NETWORK
TITLE =EA14_V41
// Act 016
// Box           : VSA14
// Input address : I96.2
// Output address: Q96.2
      CALL FC    70 (
           UnitNo                   := #UnitNo,
           ActRec                   := DB5140.EA14_V41,
           Typ                      := 1,
           FBa                      := #xTmp,
           FBa2                     := I     96.2,
           Out                      := Q     96.2);

NETWORK
TITLE =EA14_V42
// Act 017
// Box           : VSA14
// Input address : I96.3
// Output address: Q96.3
      CALL FC    70 (
           UnitNo                   := #UnitNo,
           ActRec                   := DB5140.EA14_V42,
           Typ                      := 1,
           FBa                      := #xTmp,
           FBa2                     := I     96.3,
           Out                      := Q     96.3);

NETWORK
TITLE =A14_START_MOLCH_LDT
// Act 019
// Box           : VSA14
// Output address: Q98.7
      CALL FC    70 (
           UnitNo                   := #UnitNo,
           ActRec                   := DB5140.A14_START_MOLCH_LDT,
           Typ                      := 0,
           FBa                      := #xTmp,
           FBa2                     := #xTmp,
           Out                      := Q     98.7);

NETWORK
TITLE =Molch ist unterwegs (Mixer)


      CALL FC    70 (
           UnitNo                   := #UnitNo,
           ActRec                   := DB5140.Act20,
           Typ                      := 0,
           FBa                      := #xTmp,
           FBa2                     := #xTmp,
           Out                      := Q    911.5);

NETWORK
TITLE =Molch in Endposition (Mixer)


      CALL FC    70 (
           UnitNo                   := #UnitNo,
           ActRec                   := DB5140.Act21,
           Typ                      := 0,
           FBa                      := #xTmp,
           FBa2                     := #xTmp,
           Out                      := Q    912.6);

NETWORK
TITLE =A14_POS_MOLCH
// Act 030
// Box           : VSA14
// Output address: Q98.4
      CALL FC    70 (
           UnitNo                   := #UnitNo,
           ActRec                   := DB5140.A14_POS_MOLCH,
           Typ                      := 0,
           FBa                      := #xTmp,
           FBa2                     := #xTmp,
           Out                      := Q     98.4);

NETWORK
TITLE =A14_LAUFZEIT_MOLCH
// Act 031
// Box           : VSA14
// Output address: Q98.5
      CALL FC    70 (
           UnitNo                   := #UnitNo,
           ActRec                   := DB5140.A14_LAUFZEIT_MOLCH,
           Typ                      := 0,
           FBa                      := #xTmp,
           FBa2                     := #xTmp,
           Out                      := Q     98.5);

NETWORK
TITLE =A14_TEMP_ERREICHT
// Act 032
// Box           : VSA14
// Output address: Q98.6
      CALL FC    70 (
           UnitNo                   := #UnitNo,
           ActRec                   := DB5140.A14_TEMP_ERREICHT,
           Typ                      := 0,
           FBa                      := #xTmp,
           FBa2                     := #xTmp,
           Out                      := Q     98.6);

NETWORK
TITLE =A14_Schwenkbogen  "1"=CIP  "0"=Produktion
// Act 045
// Box           : Sirup
// Output address: DB_SEND_DOEHLER.Anlage14.Schwenkbogen
      CALL FC    70 (
           UnitNo                   := #UnitNo,
           ActRec                   := DB5140.A14_Schwenkbogen,
           Typ                      := 0,
           FBa                      := #xTmp,
           FBa2                     := #xTmp,
           Out                      := DB404.DBX   67.0);

NETWORK
TITLE =A14_Molch_Sirup  "1"=Molch ist im Sirupraum
// Act 046
// Box           : Sirup
// Output address: DB_SEND_DOEHLER.Anlage14.Molch_Sirup
      CALL FC    70 (
           UnitNo                   := #UnitNo,
           ActRec                   := DB5140.A14_Molch_Sirup,
           Typ                      := 0,
           FBa                      := #xTmp,
           FBa2                     := #xTmp,
           Out                      := DB404.DBX   66.0);

NETWORK
TITLE =A14_Molch_Anlage  "1"=Molch ist an der Anlage
// Act 047
// Box           : Sirup
// Output address: DB_SEND_DOEHLER.Anlage14.Molch_Anlage
      CALL FC    70 (
           UnitNo                   := #UnitNo,
           ActRec                   := DB5140.A14_Molch_Anlage,
           Typ                      := 0,
           FBa                      := #xTmp,
           FBa2                     := #xTmp,
           Out                      := DB404.DBX   66.1);

NETWORK
TITLE =A14_Molch_PRO  "1"=Molch ist bereit für Produktion
// Act 048
// Box           : Sirup
// Output address: DB_SEND_DOEHLER.Anlage14.Molch_PRO
      CALL FC    70 (
           UnitNo                   := #UnitNo,
           ActRec                   := DB5140.A14_Molch_PRO,
           Typ                      := 0,
           FBa                      := #xTmp,
           FBa2                     := #xTmp,
           Out                      := DB404.DBX   66.2);

NETWORK
TITLE =A14_Molch_CIP  "1"=Molch ist bereit für CIP
// Act 049
// Box           : Sirup
// Output address: DB_SEND_DOEHLER.Anlage14.Molch_CIP
      CALL FC    70 (
           UnitNo                   := #UnitNo,
           ActRec                   := DB5140.A14_Molch_CIP,
           Typ                      := 0,
           FBa                      := #xTmp,
           FBa2                     := #xTmp,
           Out                      := DB404.DBX   66.3);

NETWORK
TITLE =A14_Sirupanforderung
// Act 050
// Box           : Sirup
// Output address: DB_SEND_DOEHLER.Anlage14.Sirupanforderung
      CALL FC    70 (
           UnitNo                   := #UnitNo,
           ActRec                   := DB5140.A14_Sirupanforderung,
           Typ                      := 0,
           FBa                      := #xTmp,
           FBa2                     := #xTmp,
           Out                      := DB404.DBX   66.4);

END_FUNCTION_BLOCK

FUNCTION_BLOCK FB 4141
TITLE =U114: Transfer Plant 14
FAMILY : BOTEC_F1
NAME : UniE
VERSION : 1.2


VAR_TEMP
  CIP : BOOL ;	//CIP active
  UNIM : BOOL ;	//Unit Not In Maintenance
  GenRel : BOOL ;	//general OK (emergency and maintenance OK)
  EStopOK : BOOL ;	//emergency OK
  UnitNo : INT ;	//unit number
  xTmp : BOOL ;	//Temporary Bool
  iTmp : INT ;	//Temporary INT
  rTmp : REAL ;	//Temporary REAL
  dTmp : DINT ;	//Temporary DINT (free for general use)
  RetValInt : INT ;	//return value
END_VAR
BEGIN
NETWORK
TITLE =General

      SET   ;
// Simulation ---------------------------------------------------------------
      A     DB4141.DBX 1357.7;
      CC    FB  4149; // "U114Sim"
      A     DB4141.DBX   17.3;
      =     DB4141.DBX 1357.7; //Help bit for simulation

// get unit number ----------------------------------------------------------
      L     DB4140.DBW    0;
      T     #UnitNo;

// communication ------------------------------------------------------------
      UC    FB  4145; // U114Com

NETWORK
TITLE =Sequence organisation

      CLR   ;
      =     M    122.2;

// sequencer ----------------------------------------------------------------
      A     DB4143.DBX   43.1;
      S     DB4143.DBX   97.3;

      CALL FC    40 (
           UnitNo                   := #UnitNo);

END_FUNCTION_BLOCK

FUNCTION_BLOCK FB 4210
TITLE =U121: Planung Transfer VE1
FAMILY : BOTEC_F1
NAME : U121A
VERSION : 2.1


VAR_TEMP
  EStopOK : BOOL ;	//auxiliary flag
  CIP : BOOL ;	//CIP Program Selected
  xTmp : BOOL ;	//Temporary Bool(free for general use)
  DummyBool : BOOL ;	//Temporary Bool(free for general use)
  UnitNo : INT ;	//unit number
  UnitFB : INT ;	//unit expansion FB number
  rTmp : REAL ;	//Temporary REAL (free for general use)
  iTmp : INT ;	//Temporary INT (free for general use)
  DummyInt : INT ;	//Temporary INT (free for general use)
  dTmp : DINT ;	//Temporary DINT (free for general use)
END_VAR
BEGIN
NETWORK
TITLE =general

      CLR   ;
      =     #xTmp;
      =     #EStopOK;

      L     DB4210.DBW    0;
      T     #UnitNo;
      L     DB4210.DBW    2;
      T     #UnitFB;

NETWORK
TITLE =analog inputs

      NOP   0;
// C_AnI01 AnI 001 spare
      CALL FC    24 (
           UnitNo                   := #UnitNo,
           AnIRec                   := DB5213.C_AnI01,
           ValPer                   := #DummyInt);

// C_AnI002 AnI 002 spare
      CALL FC    24 (
           UnitNo                   := #UnitNo,
           AnIRec                   := DB5213.C_AnI002,
           ValPer                   := #DummyInt);

// AnI03 AnI 003 spare
      CALL FC    24 (
           UnitNo                   := #UnitNo,
           AnIRec                   := DB5213.AnI03,
           ValPer                   := #DummyInt);

NETWORK
TITLE =Universal value

      NOP   0;
// unv001 UnV 001 Process Status
      CALL FC    27 (
           UnitNo                   := #UnitNo,
           UnVRec                   := DB5215.unv001,
           ValExt                   := DB5215.DBD  234);

// unv002 UnV 002 Universal Value 02
      CALL FC    27 (
           UnitNo                   := #UnitNo,
           UnVRec                   := DB5215.unv002,
           ValExt                   := DB5215.DBD  362);

// unv003 UnV 003 Druck Sollwert
      CALL FC    27 (
           UnitNo                   := #UnitNo,
           UnVRec                   := DB5215.unv003,
           ValExt                   := DB5215.DBD  490);

// unv004 UnV 004 Universal Value 04
      CALL FC    27 (
           UnitNo                   := #UnitNo,
           UnVRec                   := DB5215.unv004,
           ValExt                   := DB5215.DBD  618);

NETWORK
TITLE =special inputs

      NOP   0;
// SpI01 SpI 001 spare
      CALL FC    14 (
           UnitNo                   := #UnitNo,
           SpIRec                   := DB5211.SpI01,
           SpIBit                   := #DummyBool);

// SpI02 SpI 002 spare
      CALL FC    14 (
           UnitNo                   := #UnitNo,
           SpIRec                   := DB5211.SpI02,
           SpIBit                   := #DummyBool);

// SpI03 SpI 003 spare
      CALL FC    14 (
           UnitNo                   := #UnitNo,
           SpIRec                   := DB5211.SpI03,
           SpIBit                   := #DummyBool);

// SpI04 SpI 004 spare
      CALL FC    14 (
           UnitNo                   := #UnitNo,
           SpIRec                   := DB5211.SpI04,
           SpIBit                   := #DummyBool);

NETWORK
TITLE =messages

      NOP   0;
// msg001 Msg 001 Message 01
      CALL FC    16 (
           UnitNo                   := #UnitNo,
           MsgRec                   := DB5217.msg001,
           MsgBit                   := DB5217.DBX   82.7);

// msg002 Msg 002 Message 02
      CALL FC    16 (
           UnitNo                   := #UnitNo,
           MsgRec                   := DB5217.msg002,
           MsgBit                   := DB5217.DBX  142.7);

// msg003 Msg 003 Message 03
      CALL FC    16 (
           UnitNo                   := #UnitNo,
           MsgRec                   := DB5217.msg003,
           MsgBit                   := DB5217.DBX  202.7);

NETWORK
TITLE =controllers

      NOP   0;
// PID01 PID 001 spare
      CALL FC    55 (
           UnitNo                   := #UnitNo,
           PIDRec                   := DB5216.PID01,
           SpExt                    := DB5216.DBD  234,
           PVal                     := DB5216.DBD  254,
           OPer                     := #DummyInt);

NETWORK
TITLE =unit supply

      UC    FB [#UnitFB];
END_FUNCTION_BLOCK

FUNCTION_BLOCK FB 4211
TITLE =U121: Planung Transfer VE1
FAMILY : BOTEC_F1
NAME : U121E
VERSION : 1.2


VAR_TEMP
  CIP : BOOL ;	//CIP active
  UNIM : BOOL ;	//Unit Not In Maintenance
  GenRel : BOOL ;	//general OK (emergency and maintenance OK)
  EStopOK : BOOL ;	//emergency OK
  UnitNo : INT ;	//unit number
  xTmp : BOOL ;	//Temporary Bool
  iTmp : INT ;	//Temporary INT
  rTmp : REAL ;	//Temporary REAL
  dTmp : DINT ;	//Temporary DINT (free for general use)
  RetValInt : INT ;	//return value
END_VAR
BEGIN
NETWORK
TITLE =General

      SET   ;
// Simulation ---------------------------------------------------------------
      A     DB4211.DBX 1357.7;
      CC    FB  4219; // "U121Sim"
      A     DB4211.DBX   17.3;
      =     DB4211.DBX 1357.7; //Help bit for simulation

// get unit number ----------------------------------------------------------
      L     DB4210.DBW    0;
      T     #UnitNo;

// CIP ----------------------------------------------------------------------
      L     DB4211.DBD   54;
      L     0;
      <D    ;
      =     #CIP;

// emergency OK -------------------------------------------------------------
      A     DB4215.DBX   27.0; //Emergency Stop OK
      =     #EStopOK;

// Write Unit in Maintenance ------------------------------------------------

      AN    DB4211.DBX   69.7;
      =     #UNIM;

// emergency and maintenance OK ---------------------------------------------
      A     #EStopOK;
      A     #UNIM;
      =     #GenRel;

// communication ------------------------------------------------------------
      UC    FB  4215; // U121Com

NETWORK
TITLE =Analog Inputs

      NOP   0;

// ----------------------------------------------------------
// C_AnI01 spare
// ----------------------------------------------------------
      L     DB4211.DBD 1118; // !!! insert correct SFM !!!
      T     DB5213.DBD  238;

      SET   ;
      =     DB5213.DBX  141.5;

// ----------------------------------------------------------
// C_AnI002 spare
// ----------------------------------------------------------
      L     DB4211.DBD 1118; // !!! insert correct SFM !!!
      T     DB5213.DBD  358;

      SET   ;
      =     DB5213.DBX  261.5;

// ----------------------------------------------------------
// AnI03 spare
// ----------------------------------------------------------
      L     DB4211.DBD 1118; // !!! insert correct SFM !!!
      T     DB5213.DBD  478;

      SET   ;
      =     DB5213.DBX  381.5;

NETWORK
TITLE =Universal Value

      NOP   0;

// ----------------------------------------------------------
// unv001 Process Status
// ----------------------------------------------------------
// process value to UnV
//      L     0.000000e+000
//      T     "U121UnVD".unv001.ValExt

// ----------------------------------------------------------
// unv002 Universal Value 02
// ----------------------------------------------------------
// process value to UnV
//      L     0.000000e+000
//      T     "U121UnVD".unv002.ValExt

// ----------------------------------------------------------
// unv003 Druck Sollwert
// ----------------------------------------------------------
// process value to UnV
//      L     0.000000e+000
//      T     "U121UnVD".unv003.ValExt

// ----------------------------------------------------------
// unv004 Universal Value 04
// ----------------------------------------------------------
// process value to UnV
//      L     0.000000e+000
//      T     "U121UnVD".unv004.ValExt

NETWORK
TITLE =Special Input

      NOP   0;

// ----------------------------------------------------------
// SpI01 spare
// ----------------------------------------------------------
      SET   ;
      =     DB5211.DBX   81.4;
      =     DB5211.DBX   81.5;

// ----------------------------------------------------------
// SpI02 spare
// ----------------------------------------------------------
      SET   ;
      =     DB5211.DBX  141.4;
      =     DB5211.DBX  141.5;

// ----------------------------------------------------------
// SpI03 spare
// ----------------------------------------------------------
      SET   ;
      =     DB5211.DBX  201.4;
      =     DB5211.DBX  201.5;

// ----------------------------------------------------------
// SpI04 spare
// ----------------------------------------------------------
      SET   ;
      =     DB5211.DBX  261.4;
      =     DB5211.DBX  261.5;

NETWORK
TITLE =Messages

      NOP   0;

// ----------------------------------------------------------
// msg001 Message 01
// ----------------------------------------------------------
      SET   ;
      R     DB5217.DBX   80.7;
      =     DB5217.DBX   81.4;

      CLR   ;
      =     DB5217.DBX   82.7;

// ----------------------------------------------------------
// msg002 Message 02
// ----------------------------------------------------------
      SET   ;
      R     DB5217.DBX  140.7;
      =     DB5217.DBX  141.4;

      CLR   ;
      =     DB5217.DBX  142.7;

// ----------------------------------------------------------
// msg003 Message 03
// ----------------------------------------------------------
      SET   ;
      R     DB5217.DBX  200.7;
      =     DB5217.DBX  201.4;

      CLR   ;
      =     DB5217.DBX  202.7;

NETWORK
TITLE =PID controller

      NOP   0;

// ----------------------------------------------------------
// PID01 spare
// ----------------------------------------------------------
// starting value -----------------------
//A     "U121ActD".Act.OutI // !!! insert correct Act !!!
      A     #GenRel;
      CLR   ;
      =     DB5216.DBX  203.2;
      =     DB5216.DBX  203.5;

// enable alarm -------------------------
      A     DB5216.DBX  203.5;
      A     DB5216.DBX  201.4;
      AN    DB5216.DBX  203.1;
      AN    DB5216.DBX  203.3;
      AN    DB5216.DBX  203.4;
      =     DB5216.DBX  203.0;

// setpoint to controller ---------------
      L     DB4211.DBD 1118; // !!! insert correct SFM !!!
      T     DB5216.DBD  234;

// static value to controller ----------
      L     DB4211.DBD 1118; // !!! insert correct SFM !!!
      T     DB5216.DBD  238;

// process value to controller ----------
      L     DB5213.DBD   26; // !!! insert correct AnI !!!
      T     DB5216.DBD  254;

// low/high value to controller ---------
      L     DB5213.DBD   30; // !!! insert correct AnI !!!
      T     DB5216.DBD  218;

      L     DB5213.DBD   34; // !!! insert correct AnI !!!
      T     DB5216.DBD  222;

NETWORK
TITLE =Sequence organisation

      CLR   ;
      =     M    122.2;

// SFM supply ----------------------------------------------------------------

// analog value to SFM spare -----------------------
      L     DB5213.DBD  146;
      T     DB4211.DBD 1122; // !!! insert correct SFM !!!

// analog value to SFM spare -----------------------
      L     DB5213.DBD  266;
      T     DB4211.DBD 1122; // !!! insert correct SFM !!!

// analog value to SFM spare -----------------------
      L     DB5213.DBD  386;
      T     DB4211.DBD 1122; // !!! insert correct SFM !!!

// sequencer ----------------------------------------------------------------
      A     DB4213.DBX   43.1;
      S     DB4213.DBX   97.3;

      CALL FC    40 (
           UnitNo                   := #UnitNo);

NETWORK
TITLE =Auto / Manual

      SET   ;
      AN    M    122.2;
      JC    MODE;
      AN    M    120.1;


// assign PID mode
      S     DB5216.DBX  201.4;
      S     DB5216.DBX  201.5;


MODE: SET   ;

END_FUNCTION_BLOCK

FUNCTION_BLOCK FB 4220
TITLE =U122: Planung Transfer VE2
FAMILY : BOTEC_F1
NAME : U122A
VERSION : 2.1


VAR_TEMP
  EStopOK : BOOL ;	//auxiliary flag
  CIP : BOOL ;	//CIP Program Selected
  xTmp : BOOL ;	//Temporary Bool(free for general use)
  DummyBool : BOOL ;	//Temporary Bool(free for general use)
  UnitNo : INT ;	//unit number
  UnitFB : INT ;	//unit expansion FB number
  rTmp : REAL ;	//Temporary REAL (free for general use)
  iTmp : INT ;	//Temporary INT (free for general use)
  DummyInt : INT ;	//Temporary INT (free for general use)
  dTmp : DINT ;	//Temporary DINT (free for general use)
END_VAR
BEGIN
NETWORK
TITLE =general

      CLR   ;
      =     #xTmp;
      =     #EStopOK;

      L     DB4220.DBW    0;
      T     #UnitNo;
      L     DB4220.DBW    2;
      T     #UnitFB;

NETWORK
TITLE =analog inputs

      NOP   0;
// C_AnI01 AnI 001 spare
      CALL FC    24 (
           UnitNo                   := #UnitNo,
           AnIRec                   := DB5223.C_AnI01,
           ValPer                   := #DummyInt);

// C_AnI002 AnI 002 spare
      CALL FC    24 (
           UnitNo                   := #UnitNo,
           AnIRec                   := DB5223.C_AnI002,
           ValPer                   := #DummyInt);

// AnI03 AnI 003 spare
      CALL FC    24 (
           UnitNo                   := #UnitNo,
           AnIRec                   := DB5223.AnI03,
           ValPer                   := #DummyInt);

NETWORK
TITLE =Universal value

      NOP   0;
// unv001 UnV 001 Process Status
      CALL FC    27 (
           UnitNo                   := #UnitNo,
           UnVRec                   := DB5225.unv001,
           ValExt                   := DB5225.DBD  234);

// unv002 UnV 002 Universal Value 02
      CALL FC    27 (
           UnitNo                   := #UnitNo,
           UnVRec                   := DB5225.unv002,
           ValExt                   := DB5225.DBD  362);

// unv003 UnV 003 Druck Sollwert
      CALL FC    27 (
           UnitNo                   := #UnitNo,
           UnVRec                   := DB5225.unv003,
           ValExt                   := DB5225.DBD  490);

// unv004 UnV 004 Universal Value 04
      CALL FC    27 (
           UnitNo                   := #UnitNo,
           UnVRec                   := DB5225.unv004,
           ValExt                   := DB5225.DBD  618);

NETWORK
TITLE =special inputs

      NOP   0;
// SpI01 SpI 001 spare
      CALL FC    14 (
           UnitNo                   := #UnitNo,
           SpIRec                   := DB5221.SpI01,
           SpIBit                   := #DummyBool);

// SpI02 SpI 002 spare
      CALL FC    14 (
           UnitNo                   := #UnitNo,
           SpIRec                   := DB5221.SpI02,
           SpIBit                   := #DummyBool);

// SpI03 SpI 003 spare
      CALL FC    14 (
           UnitNo                   := #UnitNo,
           SpIRec                   := DB5221.SpI03,
           SpIBit                   := #DummyBool);

// SpI04 SpI 004 spare
      CALL FC    14 (
           UnitNo                   := #UnitNo,
           SpIRec                   := DB5221.SpI04,
           SpIBit                   := #DummyBool);

NETWORK
TITLE =messages

      NOP   0;
// msg001 Msg 001 Message 01
      CALL FC    16 (
           UnitNo                   := #UnitNo,
           MsgRec                   := DB5227.msg001,
           MsgBit                   := DB5227.DBX   82.7);

// msg002 Msg 002 Message 02
      CALL FC    16 (
           UnitNo                   := #UnitNo,
           MsgRec                   := DB5227.msg002,
           MsgBit                   := DB5227.DBX  142.7);

// msg003 Msg 003 Message 03
      CALL FC    16 (
           UnitNo                   := #UnitNo,
           MsgRec                   := DB5227.msg003,
           MsgBit                   := DB5227.DBX  202.7);

NETWORK
TITLE =controllers

      NOP   0;
// PID01 PID 001 spare
      CALL FC    55 (
           UnitNo                   := #UnitNo,
           PIDRec                   := DB5226.PID01,
           SpExt                    := DB5226.DBD  234,
           PVal                     := DB5226.DBD  254,
           OPer                     := #DummyInt);

NETWORK
TITLE =unit supply

      UC    FB [#UnitFB];
END_FUNCTION_BLOCK

FUNCTION_BLOCK FB 4221
TITLE =U122: Planung Transfer VE2
FAMILY : BOTEC_F1
NAME : U122E
VERSION : 1.2


VAR_TEMP
  CIP : BOOL ;	//CIP active
  UNIM : BOOL ;	//Unit Not In Maintenance
  GenRel : BOOL ;	//general OK (emergency and maintenance OK)
  EStopOK : BOOL ;	//emergency OK
  UnitNo : INT ;	//unit number
  xTmp : BOOL ;	//Temporary Bool
  iTmp : INT ;	//Temporary INT
  rTmp : REAL ;	//Temporary REAL
  dTmp : DINT ;	//Temporary DINT (free for general use)
  RetValInt : INT ;	//return value
END_VAR
BEGIN
NETWORK
TITLE =General

      SET   ;
// Simulation ---------------------------------------------------------------
      A     DB4221.DBX 1357.7;
      CC    FB  4229; // "U122Sim"
      A     DB4221.DBX   17.3;
      =     DB4221.DBX 1357.7; //Help bit for simulation

// get unit number ----------------------------------------------------------
      L     DB4220.DBW    0;
      T     #UnitNo;

// CIP ----------------------------------------------------------------------
      L     DB4221.DBD   54;
      L     0;
      <D    ;
      =     #CIP;

// emergency OK -------------------------------------------------------------
      A     DB4225.DBX   27.0; //Emergency Stop OK
      =     #EStopOK;

// Write Unit in Maintenance ------------------------------------------------

      AN    DB4221.DBX   69.7;
      =     #UNIM;

// emergency and maintenance OK ---------------------------------------------
      A     #EStopOK;
      A     #UNIM;
      =     #GenRel;

// communication ------------------------------------------------------------
      UC    FB  4225; // U122Com

NETWORK
TITLE =Analog Inputs

      NOP   0;

// ----------------------------------------------------------
// C_AnI01 spare
// ----------------------------------------------------------
      L     DB4221.DBD 1118; // !!! insert correct SFM !!!
      T     DB5223.DBD  238;

      SET   ;
      =     DB5223.DBX  141.5;

// ----------------------------------------------------------
// C_AnI002 spare
// ----------------------------------------------------------
      L     DB4221.DBD 1118; // !!! insert correct SFM !!!
      T     DB5223.DBD  358;

      SET   ;
      =     DB5223.DBX  261.5;

// ----------------------------------------------------------
// AnI03 spare
// ----------------------------------------------------------
      L     DB4221.DBD 1118; // !!! insert correct SFM !!!
      T     DB5223.DBD  478;

      SET   ;
      =     DB5223.DBX  381.5;

NETWORK
TITLE =Universal Value

      NOP   0;

// ----------------------------------------------------------
// unv001 Process Status
// ----------------------------------------------------------
// process value to UnV
//      L     0.000000e+000
//      T     "U122UnVD".unv001.ValExt

// ----------------------------------------------------------
// unv002 Universal Value 02
// ----------------------------------------------------------
// process value to UnV
//      L     0.000000e+000
//      T     "U122UnVD".unv002.ValExt

// ----------------------------------------------------------
// unv003 Druck Sollwert
// ----------------------------------------------------------
// process value to UnV
//      L     0.000000e+000
//      T     "U122UnVD".unv003.ValExt

// ----------------------------------------------------------
// unv004 Universal Value 04
// ----------------------------------------------------------
// process value to UnV
//      L     0.000000e+000
//      T     "U122UnVD".unv004.ValExt

NETWORK
TITLE =Special Input

      NOP   0;

// ----------------------------------------------------------
// SpI01 spare
// ----------------------------------------------------------
      SET   ;
      =     DB5221.DBX   81.4;
      =     DB5221.DBX   81.5;

// ----------------------------------------------------------
// SpI02 spare
// ----------------------------------------------------------
      SET   ;
      =     DB5221.DBX  141.4;
      =     DB5221.DBX  141.5;

// ----------------------------------------------------------
// SpI03 spare
// ----------------------------------------------------------
      SET   ;
      =     DB5221.DBX  201.4;
      =     DB5221.DBX  201.5;

// ----------------------------------------------------------
// SpI04 spare
// ----------------------------------------------------------
      SET   ;
      =     DB5221.DBX  261.4;
      =     DB5221.DBX  261.5;

NETWORK
TITLE =Messages

      NOP   0;

// ----------------------------------------------------------
// msg001 Message 01
// ----------------------------------------------------------
      SET   ;
      R     DB5227.DBX   80.7;
      =     DB5227.DBX   81.4;

      CLR   ;
      =     DB5227.DBX   82.7;

// ----------------------------------------------------------
// msg002 Message 02
// ----------------------------------------------------------
      SET   ;
      R     DB5227.DBX  140.7;
      =     DB5227.DBX  141.4;

      CLR   ;
      =     DB5227.DBX  142.7;

// ----------------------------------------------------------
// msg003 Message 03
// ----------------------------------------------------------
      SET   ;
      R     DB5227.DBX  200.7;
      =     DB5227.DBX  201.4;

      CLR   ;
      =     DB5227.DBX  202.7;

NETWORK
TITLE =PID controller

      NOP   0;

// ----------------------------------------------------------
// PID01 spare
// ----------------------------------------------------------
// starting value -----------------------
//A     "U122ActD".Act.OutI // !!! insert correct Act !!!
      A     #GenRel;
      CLR   ;
      =     DB5226.DBX  203.2;
      =     DB5226.DBX  203.5;

// enable alarm -------------------------
      A     DB5226.DBX  203.5;
      A     DB5226.DBX  201.4;
      AN    DB5226.DBX  203.1;
      AN    DB5226.DBX  203.3;
      AN    DB5226.DBX  203.4;
      =     DB5226.DBX  203.0;

// setpoint to controller ---------------
      L     DB4221.DBD 1118; // !!! insert correct SFM !!!
      T     DB5226.DBD  234;

// static value to controller ----------
      L     DB4221.DBD 1118; // !!! insert correct SFM !!!
      T     DB5226.DBD  238;

// process value to controller ----------
      L     DB5223.DBD   26; // !!! insert correct AnI !!!
      T     DB5226.DBD  254;

// low/high value to controller ---------
      L     DB5223.DBD   30; // !!! insert correct AnI !!!
      T     DB5226.DBD  218;

      L     DB5223.DBD   34; // !!! insert correct AnI !!!
      T     DB5226.DBD  222;

NETWORK
TITLE =Sequence organisation

      CLR   ;
      =     M    122.2;

// SFM supply ----------------------------------------------------------------

// analog value to SFM spare -----------------------
      L     DB5223.DBD  146;
      T     DB4221.DBD 1122; // !!! insert correct SFM !!!

// analog value to SFM spare -----------------------
      L     DB5223.DBD  266;
      T     DB4221.DBD 1122; // !!! insert correct SFM !!!

// analog value to SFM spare -----------------------
      L     DB5223.DBD  386;
      T     DB4221.DBD 1122; // !!! insert correct SFM !!!

// sequencer ----------------------------------------------------------------
      A     DB4223.DBX   43.1;
      S     DB4223.DBX   97.3;

      CALL FC    40 (
           UnitNo                   := #UnitNo);

NETWORK
TITLE =Auto / Manual

      SET   ;
      AN    M    122.2;
      JC    MODE;
      AN    M    120.1;


// assign PID mode
      S     DB5226.DBX  201.4;
      S     DB5226.DBX  201.5;


MODE: SET   ;

END_FUNCTION_BLOCK

FUNCTION_BLOCK FB 4250
TITLE =U125: Planung Transfer A
FAMILY : BOTEC_F1
NAME : U125A
VERSION : 2.1


VAR_TEMP
  EStopOK : BOOL ;	//auxiliary flag
  CIP : BOOL ;	//CIP Program Selected
  xTmp : BOOL ;	//Temporary Bool(free for general use)
  DummyBool : BOOL ;	//Temporary Bool(free for general use)
  UnitNo : INT ;	//unit number
  UnitFB : INT ;	//unit expansion FB number
  rTmp : REAL ;	//Temporary REAL (free for general use)
  iTmp : INT ;	//Temporary INT (free for general use)
  DummyInt : INT ;	//Temporary INT (free for general use)
  dTmp : DINT ;	//Temporary DINT (free for general use)
END_VAR
BEGIN
NETWORK
TITLE =general

      CLR   ;
      =     #xTmp;
      =     #EStopOK;

      L     DB4250.DBW    0;
      T     #UnitNo;
      L     DB4250.DBW    2;
      T     #UnitFB;

NETWORK
TITLE =analog inputs

      NOP   0;
// C_AnI01 AnI 001 spare
      CALL FC    24 (
           UnitNo                   := #UnitNo,
           AnIRec                   := DB5253.C_AnI01,
           ValPer                   := #DummyInt);

// C_AnI002 AnI 002 spare
      CALL FC    24 (
           UnitNo                   := #UnitNo,
           AnIRec                   := DB5253.C_AnI002,
           ValPer                   := #DummyInt);

// AnI03 AnI 003 spare
      CALL FC    24 (
           UnitNo                   := #UnitNo,
           AnIRec                   := DB5253.AnI03,
           ValPer                   := #DummyInt);

NETWORK
TITLE =Universal value

      NOP   0;
// unv001 UnV 001 Process Status
      CALL FC    27 (
           UnitNo                   := #UnitNo,
           UnVRec                   := DB5255.unv001,
           ValExt                   := DB5255.DBD  234);

// unv002 UnV 002 Universal Value 02
      CALL FC    27 (
           UnitNo                   := #UnitNo,
           UnVRec                   := DB5255.unv002,
           ValExt                   := DB5255.DBD  362);

// unv003 UnV 003 Druck Sollwert
      CALL FC    27 (
           UnitNo                   := #UnitNo,
           UnVRec                   := DB5255.unv003,
           ValExt                   := DB5255.DBD  490);

// unv004 UnV 004 Universal Value 04
      CALL FC    27 (
           UnitNo                   := #UnitNo,
           UnVRec                   := DB5255.unv004,
           ValExt                   := DB5255.DBD  618);

NETWORK
TITLE =special inputs

      NOP   0;
// SpI01 SpI 001 spare
      CALL FC    14 (
           UnitNo                   := #UnitNo,
           SpIRec                   := DB5251.SpI01,
           SpIBit                   := #DummyBool);

// SpI02 SpI 002 spare
      CALL FC    14 (
           UnitNo                   := #UnitNo,
           SpIRec                   := DB5251.SpI02,
           SpIBit                   := #DummyBool);

// SpI03 SpI 003 spare
      CALL FC    14 (
           UnitNo                   := #UnitNo,
           SpIRec                   := DB5251.SpI03,
           SpIBit                   := #DummyBool);

// SpI04 SpI 004 spare
      CALL FC    14 (
           UnitNo                   := #UnitNo,
           SpIRec                   := DB5251.SpI04,
           SpIBit                   := #DummyBool);

NETWORK
TITLE =messages

      NOP   0;
// msg001 Msg 001 Message 01
      CALL FC    16 (
           UnitNo                   := #UnitNo,
           MsgRec                   := DB5257.msg001,
           MsgBit                   := DB5257.DBX   82.7);

// msg002 Msg 002 Message 02
      CALL FC    16 (
           UnitNo                   := #UnitNo,
           MsgRec                   := DB5257.msg002,
           MsgBit                   := DB5257.DBX  142.7);

// msg003 Msg 003 Message 03
      CALL FC    16 (
           UnitNo                   := #UnitNo,
           MsgRec                   := DB5257.msg003,
           MsgBit                   := DB5257.DBX  202.7);

NETWORK
TITLE =controllers

      NOP   0;
// PID01 PID 001 spare
      CALL FC    55 (
           UnitNo                   := #UnitNo,
           PIDRec                   := DB5256.PID01,
           SpExt                    := DB5256.DBD  234,
           PVal                     := DB5256.DBD  254,
           OPer                     := #DummyInt);

NETWORK
TITLE =unit supply

      UC    FB [#UnitFB];
END_FUNCTION_BLOCK

FUNCTION_BLOCK FB 4251
TITLE =U125: Planung Transfer A
FAMILY : BOTEC_F1
NAME : U125E
VERSION : 1.2


VAR_TEMP
  CIP : BOOL ;	//CIP active
  UNIM : BOOL ;	//Unit Not In Maintenance
  GenRel : BOOL ;	//general OK (emergency and maintenance OK)
  EStopOK : BOOL ;	//emergency OK
  UnitNo : INT ;	//unit number
  xTmp : BOOL ;	//Temporary Bool
  iTmp : INT ;	//Temporary INT
  rTmp : REAL ;	//Temporary REAL
  dTmp : DINT ;	//Temporary DINT (free for general use)
  RetValInt : INT ;	//return value
END_VAR
BEGIN
NETWORK
TITLE =General

      SET   ;
// Simulation ---------------------------------------------------------------
      A     DB4251.DBX 1357.7;
      CC    FB  4259; // "U125Sim"
      A     DB4251.DBX   17.3;
      =     DB4251.DBX 1357.7; //Help bit for simulation

// get unit number ----------------------------------------------------------
      L     DB4250.DBW    0;
      T     #UnitNo;

// CIP ----------------------------------------------------------------------
      L     DB4251.DBD   54;
      L     0;
      <D    ;
      =     #CIP;

// emergency OK -------------------------------------------------------------
      A     DB4255.DBX   27.0; //Emergency Stop OK
      =     #EStopOK;

// Write Unit in Maintenance ------------------------------------------------

      AN    DB4251.DBX   69.7;
      =     #UNIM;

// emergency and maintenance OK ---------------------------------------------
      A     #EStopOK;
      A     #UNIM;
      =     #GenRel;

// communication ------------------------------------------------------------
      UC    FB  4255; // U125Com

NETWORK
TITLE =Analog Inputs

      NOP   0;

// ----------------------------------------------------------
// C_AnI01 spare
// ----------------------------------------------------------
      L     DB4251.DBD 1118; // !!! insert correct SFM !!!
      T     DB5253.DBD  238;

      SET   ;
      =     DB5253.DBX  141.5;

// ----------------------------------------------------------
// C_AnI002 spare
// ----------------------------------------------------------
      L     DB4251.DBD 1118; // !!! insert correct SFM !!!
      T     DB5253.DBD  358;

      SET   ;
      =     DB5253.DBX  261.5;

// ----------------------------------------------------------
// AnI03 spare
// ----------------------------------------------------------
      L     DB4251.DBD 1118; // !!! insert correct SFM !!!
      T     DB5253.DBD  478;

      SET   ;
      =     DB5253.DBX  381.5;

NETWORK
TITLE =Universal Value

      NOP   0;

// ----------------------------------------------------------
// unv001 Process Status
// ----------------------------------------------------------
// process value to UnV
//      L     0.000000e+000
//      T     "U125UnVD".unv001.ValExt

// ----------------------------------------------------------
// unv002 Universal Value 02
// ----------------------------------------------------------
// process value to UnV
//      L     0.000000e+000
//      T     "U125UnVD".unv002.ValExt

// ----------------------------------------------------------
// unv003 Druck Sollwert
// ----------------------------------------------------------
// process value to UnV
//      L     0.000000e+000
//      T     "U125UnVD".unv003.ValExt

// ----------------------------------------------------------
// unv004 Universal Value 04
// ----------------------------------------------------------
// process value to UnV
//      L     0.000000e+000
//      T     "U125UnVD".unv004.ValExt

NETWORK
TITLE =Special Input

      NOP   0;

// ----------------------------------------------------------
// SpI01 spare
// ----------------------------------------------------------
      SET   ;
      =     DB5251.DBX   81.4;
      =     DB5251.DBX   81.5;

// ----------------------------------------------------------
// SpI02 spare
// ----------------------------------------------------------
      SET   ;
      =     DB5251.DBX  141.4;
      =     DB5251.DBX  141.5;

// ----------------------------------------------------------
// SpI03 spare
// ----------------------------------------------------------
      SET   ;
      =     DB5251.DBX  201.4;
      =     DB5251.DBX  201.5;

// ----------------------------------------------------------
// SpI04 spare
// ----------------------------------------------------------
      SET   ;
      =     DB5251.DBX  261.4;
      =     DB5251.DBX  261.5;

NETWORK
TITLE =Messages

      NOP   0;

// ----------------------------------------------------------
// msg001 Message 01
// ----------------------------------------------------------
      SET   ;
      R     DB5257.DBX   80.7;
      =     DB5257.DBX   81.4;

      CLR   ;
      =     DB5257.DBX   82.7;

// ----------------------------------------------------------
// msg002 Message 02
// ----------------------------------------------------------
      SET   ;
      R     DB5257.DBX  140.7;
      =     DB5257.DBX  141.4;

      CLR   ;
      =     DB5257.DBX  142.7;

// ----------------------------------------------------------
// msg003 Message 03
// ----------------------------------------------------------
      SET   ;
      R     DB5257.DBX  200.7;
      =     DB5257.DBX  201.4;

      CLR   ;
      =     DB5257.DBX  202.7;

NETWORK
TITLE =PID controller

      NOP   0;

// ----------------------------------------------------------
// PID01 spare
// ----------------------------------------------------------
// starting value -----------------------
//A     "U125ActD".Act.OutI // !!! insert correct Act !!!
      A     #GenRel;
      CLR   ;
      =     DB5256.DBX  203.2;
      =     DB5256.DBX  203.5;

// enable alarm -------------------------
      A     DB5256.DBX  203.5;
      A     DB5256.DBX  201.4;
      AN    DB5256.DBX  203.1;
      AN    DB5256.DBX  203.3;
      AN    DB5256.DBX  203.4;
      =     DB5256.DBX  203.0;

// setpoint to controller ---------------
      L     DB4251.DBD 1118; // !!! insert correct SFM !!!
      T     DB5256.DBD  234;

// static value to controller ----------
      L     DB4251.DBD 1118; // !!! insert correct SFM !!!
      T     DB5256.DBD  238;

// process value to controller ----------
      L     DB5253.DBD   26; // !!! insert correct AnI !!!
      T     DB5256.DBD  254;

// low/high value to controller ---------
      L     DB5253.DBD   30; // !!! insert correct AnI !!!
      T     DB5256.DBD  218;

      L     DB5253.DBD   34; // !!! insert correct AnI !!!
      T     DB5256.DBD  222;

NETWORK
TITLE =Sequence organisation

      CLR   ;
      =     M    122.2;

// SFM supply ----------------------------------------------------------------

// analog value to SFM spare -----------------------
      L     DB5253.DBD  146;
      T     DB4251.DBD 1122; // !!! insert correct SFM !!!

// analog value to SFM spare -----------------------
      L     DB5253.DBD  266;
      T     DB4251.DBD 1122; // !!! insert correct SFM !!!

// analog value to SFM spare -----------------------
      L     DB5253.DBD  386;
      T     DB4251.DBD 1122; // !!! insert correct SFM !!!

// sequencer ----------------------------------------------------------------
      A     DB4253.DBX   43.1;
      S     DB4253.DBX   97.3;

      CALL FC    40 (
           UnitNo                   := #UnitNo);

NETWORK
TITLE =Auto / Manual

      SET   ;
      AN    M    122.2;
      JC    MODE;
      AN    M    120.1;


// assign PID mode
      S     DB5256.DBX  201.4;
      S     DB5256.DBX  201.5;


MODE: SET   ;

END_FUNCTION_BLOCK

FUNCTION_BLOCK FB 4260
TITLE =U126: Planung Transfer B
FAMILY : BOTEC_F1
NAME : U126A
VERSION : 2.1


VAR_TEMP
  EStopOK : BOOL ;	//auxiliary flag
  CIP : BOOL ;	//CIP Program Selected
  xTmp : BOOL ;	//Temporary Bool(free for general use)
  DummyBool : BOOL ;	//Temporary Bool(free for general use)
  UnitNo : INT ;	//unit number
  UnitFB : INT ;	//unit expansion FB number
  rTmp : REAL ;	//Temporary REAL (free for general use)
  iTmp : INT ;	//Temporary INT (free for general use)
  DummyInt : INT ;	//Temporary INT (free for general use)
  dTmp : DINT ;	//Temporary DINT (free for general use)
END_VAR
BEGIN
NETWORK
TITLE =general

      CLR   ;
      =     #xTmp;
      =     #EStopOK;

      L     DB4260.DBW    0;
      T     #UnitNo;
      L     DB4260.DBW    2;
      T     #UnitFB;

NETWORK
TITLE =analog inputs

      NOP   0;
// C_AnI01 AnI 001 spare
      CALL FC    24 (
           UnitNo                   := #UnitNo,
           AnIRec                   := DB5263.C_AnI01,
           ValPer                   := #DummyInt);

// C_AnI002 AnI 002 spare
      CALL FC    24 (
           UnitNo                   := #UnitNo,
           AnIRec                   := DB5263.C_AnI002,
           ValPer                   := #DummyInt);

// AnI03 AnI 003 spare
      CALL FC    24 (
           UnitNo                   := #UnitNo,
           AnIRec                   := DB5263.AnI03,
           ValPer                   := #DummyInt);

NETWORK
TITLE =Universal value

      NOP   0;
// unv001 UnV 001 Process Status
      CALL FC    27 (
           UnitNo                   := #UnitNo,
           UnVRec                   := DB5265.unv001,
           ValExt                   := DB5265.DBD  234);

// unv002 UnV 002 Universal Value 02
      CALL FC    27 (
           UnitNo                   := #UnitNo,
           UnVRec                   := DB5265.unv002,
           ValExt                   := DB5265.DBD  362);

// unv003 UnV 003 Druck Sollwert
      CALL FC    27 (
           UnitNo                   := #UnitNo,
           UnVRec                   := DB5265.unv003,
           ValExt                   := DB5265.DBD  490);

// unv004 UnV 004 Universal Value 04
      CALL FC    27 (
           UnitNo                   := #UnitNo,
           UnVRec                   := DB5265.unv004,
           ValExt                   := DB5265.DBD  618);

NETWORK
TITLE =special inputs

      NOP   0;
// SpI01 SpI 001 spare
      CALL FC    14 (
           UnitNo                   := #UnitNo,
           SpIRec                   := DB5261.SpI01,
           SpIBit                   := #DummyBool);

// SpI02 SpI 002 spare
      CALL FC    14 (
           UnitNo                   := #UnitNo,
           SpIRec                   := DB5261.SpI02,
           SpIBit                   := #DummyBool);

// SpI03 SpI 003 spare
      CALL FC    14 (
           UnitNo                   := #UnitNo,
           SpIRec                   := DB5261.SpI03,
           SpIBit                   := #DummyBool);

// SpI04 SpI 004 spare
      CALL FC    14 (
           UnitNo                   := #UnitNo,
           SpIRec                   := DB5261.SpI04,
           SpIBit                   := #DummyBool);

NETWORK
TITLE =messages

      NOP   0;
// msg001 Msg 001 Message 01
      CALL FC    16 (
           UnitNo                   := #UnitNo,
           MsgRec                   := DB5267.msg001,
           MsgBit                   := DB5267.DBX   82.7);

// msg002 Msg 002 Message 02
      CALL FC    16 (
           UnitNo                   := #UnitNo,
           MsgRec                   := DB5267.msg002,
           MsgBit                   := DB5267.DBX  142.7);

// msg003 Msg 003 Message 03
      CALL FC    16 (
           UnitNo                   := #UnitNo,
           MsgRec                   := DB5267.msg003,
           MsgBit                   := DB5267.DBX  202.7);

NETWORK
TITLE =controllers

      NOP   0;
// PID01 PID 001 spare
      CALL FC    55 (
           UnitNo                   := #UnitNo,
           PIDRec                   := DB5266.PID01,
           SpExt                    := DB5266.DBD  234,
           PVal                     := DB5266.DBD  254,
           OPer                     := #DummyInt);

NETWORK
TITLE =unit supply

      UC    FB [#UnitFB];
END_FUNCTION_BLOCK

FUNCTION_BLOCK FB 4261
TITLE =U126: Planung Transfer B
FAMILY : BOTEC_F1
NAME : U126E
VERSION : 1.2


VAR_TEMP
  CIP : BOOL ;	//CIP active
  UNIM : BOOL ;	//Unit Not In Maintenance
  GenRel : BOOL ;	//general OK (emergency and maintenance OK)
  EStopOK : BOOL ;	//emergency OK
  UnitNo : INT ;	//unit number
  xTmp : BOOL ;	//Temporary Bool
  iTmp : INT ;	//Temporary INT
  rTmp : REAL ;	//Temporary REAL
  dTmp : DINT ;	//Temporary DINT (free for general use)
  RetValInt : INT ;	//return value
END_VAR
BEGIN
NETWORK
TITLE =General

      SET   ;
// Simulation ---------------------------------------------------------------
      A     DB4261.DBX 1357.7;
      CC    FB  4269; // "U126Sim"
      A     DB4261.DBX   17.3;
      =     DB4261.DBX 1357.7; //Help bit for simulation

// get unit number ----------------------------------------------------------
      L     DB4260.DBW    0;
      T     #UnitNo;

// CIP ----------------------------------------------------------------------
      L     DB4261.DBD   54;
      L     0;
      <D    ;
      =     #CIP;

// emergency OK -------------------------------------------------------------
      A     DB4265.DBX   27.0; //Emergency Stop OK
      =     #EStopOK;

// Write Unit in Maintenance ------------------------------------------------

      AN    DB4261.DBX   69.7;
      =     #UNIM;

// emergency and maintenance OK ---------------------------------------------
      A     #EStopOK;
      A     #UNIM;
      =     #GenRel;

// communication ------------------------------------------------------------
      UC    FB  4265; // U126Com

NETWORK
TITLE =Analog Inputs

      NOP   0;

// ----------------------------------------------------------
// C_AnI01 spare
// ----------------------------------------------------------
      L     DB4261.DBD 1118; // !!! insert correct SFM !!!
      T     DB5263.DBD  238;

      SET   ;
      =     DB5263.DBX  141.5;

// ----------------------------------------------------------
// C_AnI002 spare
// ----------------------------------------------------------
      L     DB4261.DBD 1118; // !!! insert correct SFM !!!
      T     DB5263.DBD  358;

      SET   ;
      =     DB5263.DBX  261.5;

// ----------------------------------------------------------
// AnI03 spare
// ----------------------------------------------------------
      L     DB4261.DBD 1118; // !!! insert correct SFM !!!
      T     DB5263.DBD  478;

      SET   ;
      =     DB5263.DBX  381.5;

NETWORK
TITLE =Universal Value

      NOP   0;

// ----------------------------------------------------------
// unv001 Process Status
// ----------------------------------------------------------
// process value to UnV
//      L     0.000000e+000
//      T     "U126UnVD".unv001.ValExt

// ----------------------------------------------------------
// unv002 Universal Value 02
// ----------------------------------------------------------
// process value to UnV
//      L     0.000000e+000
//      T     "U126UnVD".unv002.ValExt

// ----------------------------------------------------------
// unv003 Druck Sollwert
// ----------------------------------------------------------
// process value to UnV
//      L     0.000000e+000
//      T     "U126UnVD".unv003.ValExt

// ----------------------------------------------------------
// unv004 Universal Value 04
// ----------------------------------------------------------
// process value to UnV
//      L     0.000000e+000
//      T     "U126UnVD".unv004.ValExt

NETWORK
TITLE =Special Input

      NOP   0;

// ----------------------------------------------------------
// SpI01 spare
// ----------------------------------------------------------
      SET   ;
      =     DB5261.DBX   81.4;
      =     DB5261.DBX   81.5;

// ----------------------------------------------------------
// SpI02 spare
// ----------------------------------------------------------
      SET   ;
      =     DB5261.DBX  141.4;
      =     DB5261.DBX  141.5;

// ----------------------------------------------------------
// SpI03 spare
// ----------------------------------------------------------
      SET   ;
      =     DB5261.DBX  201.4;
      =     DB5261.DBX  201.5;

// ----------------------------------------------------------
// SpI04 spare
// ----------------------------------------------------------
      SET   ;
      =     DB5261.DBX  261.4;
      =     DB5261.DBX  261.5;

NETWORK
TITLE =Messages

      NOP   0;

// ----------------------------------------------------------
// msg001 Message 01
// ----------------------------------------------------------
      SET   ;
      R     DB5267.DBX   80.7;
      =     DB5267.DBX   81.4;

      CLR   ;
      =     DB5267.DBX   82.7;

// ----------------------------------------------------------
// msg002 Message 02
// ----------------------------------------------------------
      SET   ;
      R     DB5267.DBX  140.7;
      =     DB5267.DBX  141.4;

      CLR   ;
      =     DB5267.DBX  142.7;

// ----------------------------------------------------------
// msg003 Message 03
// ----------------------------------------------------------
      SET   ;
      R     DB5267.DBX  200.7;
      =     DB5267.DBX  201.4;

      CLR   ;
      =     DB5267.DBX  202.7;

NETWORK
TITLE =PID controller

      NOP   0;

// ----------------------------------------------------------
// PID01 spare
// ----------------------------------------------------------
// starting value -----------------------
//A     "U126ActD".Act.OutI // !!! insert correct Act !!!
      A     #GenRel;
      CLR   ;
      =     DB5266.DBX  203.2;
      =     DB5266.DBX  203.5;

// enable alarm -------------------------
      A     DB5266.DBX  203.5;
      A     DB5266.DBX  201.4;
      AN    DB5266.DBX  203.1;
      AN    DB5266.DBX  203.3;
      AN    DB5266.DBX  203.4;
      =     DB5266.DBX  203.0;

// setpoint to controller ---------------
      L     DB4261.DBD 1118; // !!! insert correct SFM !!!
      T     DB5266.DBD  234;

// static value to controller ----------
      L     DB4261.DBD 1118; // !!! insert correct SFM !!!
      T     DB5266.DBD  238;

// process value to controller ----------
      L     DB5263.DBD   26; // !!! insert correct AnI !!!
      T     DB5266.DBD  254;

// low/high value to controller ---------
      L     DB5263.DBD   30; // !!! insert correct AnI !!!
      T     DB5266.DBD  218;

      L     DB5263.DBD   34; // !!! insert correct AnI !!!
      T     DB5266.DBD  222;

NETWORK
TITLE =Sequence organisation

      CLR   ;
      =     M    122.2;

// SFM supply ----------------------------------------------------------------

// analog value to SFM spare -----------------------
      L     DB5263.DBD  146;
      T     DB4261.DBD 1122; // !!! insert correct SFM !!!

// analog value to SFM spare -----------------------
      L     DB5263.DBD  266;
      T     DB4261.DBD 1122; // !!! insert correct SFM !!!

// analog value to SFM spare -----------------------
      L     DB5263.DBD  386;
      T     DB4261.DBD 1122; // !!! insert correct SFM !!!

// sequencer ----------------------------------------------------------------
      A     DB4263.DBX   43.1;
      S     DB4263.DBX   97.3;

      CALL FC    40 (
           UnitNo                   := #UnitNo);

NETWORK
TITLE =Auto / Manual

      SET   ;
      AN    M    122.2;
      JC    MODE;
      AN    M    120.1;


// assign PID mode
      S     DB5266.DBX  201.4;
      S     DB5266.DBX  201.5;


MODE: SET   ;

END_FUNCTION_BLOCK

FUNCTION_BLOCK FB 4270
TITLE =U127: Planung Transfer CF
FAMILY : BOTEC_F1
NAME : U127A
VERSION : 2.1


VAR_TEMP
  EStopOK : BOOL ;	//auxiliary flag
  CIP : BOOL ;	//CIP Program Selected
  xTmp : BOOL ;	//Temporary Bool(free for general use)
  DummyBool : BOOL ;	//Temporary Bool(free for general use)
  UnitNo : INT ;	//unit number
  UnitFB : INT ;	//unit expansion FB number
  rTmp : REAL ;	//Temporary REAL (free for general use)
  iTmp : INT ;	//Temporary INT (free for general use)
  DummyInt : INT ;	//Temporary INT (free for general use)
  dTmp : DINT ;	//Temporary DINT (free for general use)
END_VAR
BEGIN
NETWORK
TITLE =general

      CLR   ;
      =     #xTmp;
      =     #EStopOK;

      L     DB4270.DBW    0;
      T     #UnitNo;
      L     DB4270.DBW    2;
      T     #UnitFB;

NETWORK
TITLE =analog inputs

      NOP   0;
// C_AnI01 AnI 001 spare
      CALL FC    24 (
           UnitNo                   := #UnitNo,
           AnIRec                   := DB5273.C_AnI01,
           ValPer                   := #DummyInt);

// C_AnI002 AnI 002 spare
      CALL FC    24 (
           UnitNo                   := #UnitNo,
           AnIRec                   := DB5273.C_AnI002,
           ValPer                   := #DummyInt);

// AnI03 AnI 003 spare
      CALL FC    24 (
           UnitNo                   := #UnitNo,
           AnIRec                   := DB5273.AnI03,
           ValPer                   := #DummyInt);

NETWORK
TITLE =Universal value

      NOP   0;
// unv001 UnV 001 Process Status
      CALL FC    27 (
           UnitNo                   := #UnitNo,
           UnVRec                   := DB5275.unv001,
           ValExt                   := DB5275.DBD  234);

// unv002 UnV 002 Universal Value 02
      CALL FC    27 (
           UnitNo                   := #UnitNo,
           UnVRec                   := DB5275.unv002,
           ValExt                   := DB5275.DBD  362);

// unv003 UnV 003 Druck Sollwert
      CALL FC    27 (
           UnitNo                   := #UnitNo,
           UnVRec                   := DB5275.unv003,
           ValExt                   := DB5275.DBD  490);

// unv004 UnV 004 Universal Value 04
      CALL FC    27 (
           UnitNo                   := #UnitNo,
           UnVRec                   := DB5275.unv004,
           ValExt                   := DB5275.DBD  618);

NETWORK
TITLE =special inputs

      NOP   0;
// SpI01 SpI 001 spare
      CALL FC    14 (
           UnitNo                   := #UnitNo,
           SpIRec                   := DB5271.SpI01,
           SpIBit                   := #DummyBool);

// SpI02 SpI 002 spare
      CALL FC    14 (
           UnitNo                   := #UnitNo,
           SpIRec                   := DB5271.SpI02,
           SpIBit                   := #DummyBool);

// SpI03 SpI 003 spare
      CALL FC    14 (
           UnitNo                   := #UnitNo,
           SpIRec                   := DB5271.SpI03,
           SpIBit                   := #DummyBool);

// SpI04 SpI 004 spare
      CALL FC    14 (
           UnitNo                   := #UnitNo,
           SpIRec                   := DB5271.SpI04,
           SpIBit                   := #DummyBool);

NETWORK
TITLE =messages

      NOP   0;
// msg001 Msg 001 Message 01
      CALL FC    16 (
           UnitNo                   := #UnitNo,
           MsgRec                   := DB5277.msg001,
           MsgBit                   := DB5277.DBX   82.7);

// msg002 Msg 002 Message 02
      CALL FC    16 (
           UnitNo                   := #UnitNo,
           MsgRec                   := DB5277.msg002,
           MsgBit                   := DB5277.DBX  142.7);

// msg003 Msg 003 Message 03
      CALL FC    16 (
           UnitNo                   := #UnitNo,
           MsgRec                   := DB5277.msg003,
           MsgBit                   := DB5277.DBX  202.7);

NETWORK
TITLE =controllers

      NOP   0;
// PID01 PID 001 spare
      CALL FC    55 (
           UnitNo                   := #UnitNo,
           PIDRec                   := DB5276.PID01,
           SpExt                    := DB5276.DBD  234,
           PVal                     := DB5276.DBD  254,
           OPer                     := #DummyInt);

NETWORK
TITLE =unit supply

      UC    FB [#UnitFB];
END_FUNCTION_BLOCK

FUNCTION_BLOCK FB 4271
TITLE =U127: Planung Transfer CF
FAMILY : BOTEC_F1
NAME : U127E
VERSION : 1.2


VAR_TEMP
  CIP : BOOL ;	//CIP active
  UNIM : BOOL ;	//Unit Not In Maintenance
  GenRel : BOOL ;	//general OK (emergency and maintenance OK)
  EStopOK : BOOL ;	//emergency OK
  UnitNo : INT ;	//unit number
  xTmp : BOOL ;	//Temporary Bool
  iTmp : INT ;	//Temporary INT
  rTmp : REAL ;	//Temporary REAL
  dTmp : DINT ;	//Temporary DINT (free for general use)
  RetValInt : INT ;	//return value
END_VAR
BEGIN
NETWORK
TITLE =General

      SET   ;
// Simulation ---------------------------------------------------------------
      A     DB4271.DBX 1357.7;
      CC    FB  4279; // "U127Sim"
      A     DB4271.DBX   17.3;
      =     DB4271.DBX 1357.7; //Help bit for simulation

// get unit number ----------------------------------------------------------
      L     DB4270.DBW    0;
      T     #UnitNo;

// CIP ----------------------------------------------------------------------
      L     DB4271.DBD   54;
      L     0;
      <D    ;
      =     #CIP;

// emergency OK -------------------------------------------------------------
      A     DB4275.DBX   27.0; //Emergency Stop OK
      =     #EStopOK;

// Write Unit in Maintenance ------------------------------------------------

      AN    DB4271.DBX   69.7;
      =     #UNIM;

// emergency and maintenance OK ---------------------------------------------
      A     #EStopOK;
      A     #UNIM;
      =     #GenRel;

// communication ------------------------------------------------------------
      UC    FB  4275; // U127Com

NETWORK
TITLE =Analog Inputs

      NOP   0;

// ----------------------------------------------------------
// C_AnI01 spare
// ----------------------------------------------------------
      L     DB4271.DBD 1118; // !!! insert correct SFM !!!
      T     DB5273.DBD  238;

      SET   ;
      =     DB5273.DBX  141.5;

// ----------------------------------------------------------
// C_AnI002 spare
// ----------------------------------------------------------
      L     DB4271.DBD 1118; // !!! insert correct SFM !!!
      T     DB5273.DBD  358;

      SET   ;
      =     DB5273.DBX  261.5;

// ----------------------------------------------------------
// AnI03 spare
// ----------------------------------------------------------
      L     DB4271.DBD 1118; // !!! insert correct SFM !!!
      T     DB5273.DBD  478;

      SET   ;
      =     DB5273.DBX  381.5;

NETWORK
TITLE =Universal Value

      NOP   0;

// ----------------------------------------------------------
// unv001 Process Status
// ----------------------------------------------------------
// process value to UnV
//      L     0.000000e+000
//      T     "U127UnVD".unv001.ValExt

// ----------------------------------------------------------
// unv002 Universal Value 02
// ----------------------------------------------------------
// process value to UnV
//      L     0.000000e+000
//      T     "U127UnVD".unv002.ValExt

// ----------------------------------------------------------
// unv003 Druck Sollwert
// ----------------------------------------------------------
// process value to UnV
//      L     0.000000e+000
//      T     "U127UnVD".unv003.ValExt

// ----------------------------------------------------------
// unv004 Universal Value 04
// ----------------------------------------------------------
// process value to UnV
//      L     0.000000e+000
//      T     "U127UnVD".unv004.ValExt

NETWORK
TITLE =Special Input

      NOP   0;

// ----------------------------------------------------------
// SpI01 spare
// ----------------------------------------------------------
      SET   ;
      =     DB5271.DBX   81.4;
      =     DB5271.DBX   81.5;

// ----------------------------------------------------------
// SpI02 spare
// ----------------------------------------------------------
      SET   ;
      =     DB5271.DBX  141.4;
      =     DB5271.DBX  141.5;

// ----------------------------------------------------------
// SpI03 spare
// ----------------------------------------------------------
      SET   ;
      =     DB5271.DBX  201.4;
      =     DB5271.DBX  201.5;

// ----------------------------------------------------------
// SpI04 spare
// ----------------------------------------------------------
      SET   ;
      =     DB5271.DBX  261.4;
      =     DB5271.DBX  261.5;

NETWORK
TITLE =Messages

      NOP   0;

// ----------------------------------------------------------
// msg001 Message 01
// ----------------------------------------------------------
      SET   ;
      R     DB5277.DBX   80.7;
      =     DB5277.DBX   81.4;

      CLR   ;
      =     DB5277.DBX   82.7;

// ----------------------------------------------------------
// msg002 Message 02
// ----------------------------------------------------------
      SET   ;
      R     DB5277.DBX  140.7;
      =     DB5277.DBX  141.4;

      CLR   ;
      =     DB5277.DBX  142.7;

// ----------------------------------------------------------
// msg003 Message 03
// ----------------------------------------------------------
      SET   ;
      R     DB5277.DBX  200.7;
      =     DB5277.DBX  201.4;

      CLR   ;
      =     DB5277.DBX  202.7;

NETWORK
TITLE =PID controller

      NOP   0;

// ----------------------------------------------------------
// PID01 spare
// ----------------------------------------------------------
// starting value -----------------------
//A     "U127ActD".Act.OutI // !!! insert correct Act !!!
      A     #GenRel;
      CLR   ;
      =     DB5276.DBX  203.2;
      =     DB5276.DBX  203.5;

// enable alarm -------------------------
      A     DB5276.DBX  203.5;
      A     DB5276.DBX  201.4;
      AN    DB5276.DBX  203.1;
      AN    DB5276.DBX  203.3;
      AN    DB5276.DBX  203.4;
      =     DB5276.DBX  203.0;

// setpoint to controller ---------------
      L     DB4271.DBD 1118; // !!! insert correct SFM !!!
      T     DB5276.DBD  234;

// static value to controller ----------
      L     DB4271.DBD 1118; // !!! insert correct SFM !!!
      T     DB5276.DBD  238;

// process value to controller ----------
      L     DB5273.DBD   26; // !!! insert correct AnI !!!
      T     DB5276.DBD  254;

// low/high value to controller ---------
      L     DB5273.DBD   30; // !!! insert correct AnI !!!
      T     DB5276.DBD  218;

      L     DB5273.DBD   34; // !!! insert correct AnI !!!
      T     DB5276.DBD  222;

NETWORK
TITLE =Sequence organisation

      CLR   ;
      =     M    122.2;

// SFM supply ----------------------------------------------------------------

// analog value to SFM spare -----------------------
      L     DB5273.DBD  146;
      T     DB4271.DBD 1122; // !!! insert correct SFM !!!

// analog value to SFM spare -----------------------
      L     DB5273.DBD  266;
      T     DB4271.DBD 1122; // !!! insert correct SFM !!!

// analog value to SFM spare -----------------------
      L     DB5273.DBD  386;
      T     DB4271.DBD 1122; // !!! insert correct SFM !!!

// sequencer ----------------------------------------------------------------
      A     DB4273.DBX   43.1;
      S     DB4273.DBX   97.3;

      CALL FC    40 (
           UnitNo                   := #UnitNo);

NETWORK
TITLE =Auto / Manual

      SET   ;
      AN    M    122.2;
      JC    MODE;
      AN    M    120.1;


// assign PID mode
      S     DB5276.DBX  201.4;
      S     DB5276.DBX  201.5;


MODE: SET   ;

END_FUNCTION_BLOCK

FUNCTION_BLOCK FB 4280
TITLE =U128: Planung Transfer C.1
FAMILY : BOTEC_F1
NAME : U128A
VERSION : 2.1


VAR_TEMP
  EStopOK : BOOL ;	//auxiliary flag
  CIP : BOOL ;	//CIP Program Selected
  xTmp : BOOL ;	//Temporary Bool(free for general use)
  DummyBool : BOOL ;	//Temporary Bool(free for general use)
  UnitNo : INT ;	//unit number
  UnitFB : INT ;	//unit expansion FB number
  rTmp : REAL ;	//Temporary REAL (free for general use)
  iTmp : INT ;	//Temporary INT (free for general use)
  DummyInt : INT ;	//Temporary INT (free for general use)
  dTmp : DINT ;	//Temporary DINT (free for general use)
END_VAR
BEGIN
NETWORK
TITLE =general

      CLR   ;
      =     #xTmp;
      =     #EStopOK;

      L     DB4280.DBW    0;
      T     #UnitNo;
      L     DB4280.DBW    2;
      T     #UnitFB;

NETWORK
TITLE =analog inputs

      NOP   0;
// C_AnI01 AnI 001 spare
      CALL FC    24 (
           UnitNo                   := #UnitNo,
           AnIRec                   := DB5283.C_AnI01,
           ValPer                   := #DummyInt);

// C_AnI002 AnI 002 spare
      CALL FC    24 (
           UnitNo                   := #UnitNo,
           AnIRec                   := DB5283.C_AnI002,
           ValPer                   := #DummyInt);

// AnI03 AnI 003 spare
      CALL FC    24 (
           UnitNo                   := #UnitNo,
           AnIRec                   := DB5283.AnI03,
           ValPer                   := #DummyInt);

NETWORK
TITLE =Universal value

      NOP   0;
// unv001 UnV 001 Process Status
      CALL FC    27 (
           UnitNo                   := #UnitNo,
           UnVRec                   := DB5285.unv001,
           ValExt                   := DB5285.DBD  234);

// unv002 UnV 002 Universal Value 02
      CALL FC    27 (
           UnitNo                   := #UnitNo,
           UnVRec                   := DB5285.unv002,
           ValExt                   := DB5285.DBD  362);

// unv003 UnV 003 Druck Sollwert
      CALL FC    27 (
           UnitNo                   := #UnitNo,
           UnVRec                   := DB5285.unv003,
           ValExt                   := DB5285.DBD  490);

// unv004 UnV 004 Universal Value 04
      CALL FC    27 (
           UnitNo                   := #UnitNo,
           UnVRec                   := DB5285.unv004,
           ValExt                   := DB5285.DBD  618);

NETWORK
TITLE =special inputs

      NOP   0;
// SpI01 SpI 001 spare
      CALL FC    14 (
           UnitNo                   := #UnitNo,
           SpIRec                   := DB5281.SpI01,
           SpIBit                   := #DummyBool);

// SpI02 SpI 002 spare
      CALL FC    14 (
           UnitNo                   := #UnitNo,
           SpIRec                   := DB5281.SpI02,
           SpIBit                   := #DummyBool);

// SpI03 SpI 003 spare
      CALL FC    14 (
           UnitNo                   := #UnitNo,
           SpIRec                   := DB5281.SpI03,
           SpIBit                   := #DummyBool);

// SpI04 SpI 004 spare
      CALL FC    14 (
           UnitNo                   := #UnitNo,
           SpIRec                   := DB5281.SpI04,
           SpIBit                   := #DummyBool);

NETWORK
TITLE =messages

      NOP   0;
// msg001 Msg 001 Message 01
      CALL FC    16 (
           UnitNo                   := #UnitNo,
           MsgRec                   := DB5287.msg001,
           MsgBit                   := DB5287.DBX   82.7);

// msg002 Msg 002 Message 02
      CALL FC    16 (
           UnitNo                   := #UnitNo,
           MsgRec                   := DB5287.msg002,
           MsgBit                   := DB5287.DBX  142.7);

// msg003 Msg 003 Message 03
      CALL FC    16 (
           UnitNo                   := #UnitNo,
           MsgRec                   := DB5287.msg003,
           MsgBit                   := DB5287.DBX  202.7);

NETWORK
TITLE =controllers

      NOP   0;
// PID01 PID 001 spare
      CALL FC    55 (
           UnitNo                   := #UnitNo,
           PIDRec                   := DB5286.PID01,
           SpExt                    := DB5286.DBD  234,
           PVal                     := DB5286.DBD  254,
           OPer                     := #DummyInt);

NETWORK
TITLE =unit supply

      UC    FB [#UnitFB];
END_FUNCTION_BLOCK

FUNCTION_BLOCK FB 4281
TITLE =U128: Planung Transfer C.1
FAMILY : BOTEC_F1
NAME : U128E
VERSION : 1.2


VAR_TEMP
  CIP : BOOL ;	//CIP active
  UNIM : BOOL ;	//Unit Not In Maintenance
  GenRel : BOOL ;	//general OK (emergency and maintenance OK)
  EStopOK : BOOL ;	//emergency OK
  UnitNo : INT ;	//unit number
  xTmp : BOOL ;	//Temporary Bool
  iTmp : INT ;	//Temporary INT
  rTmp : REAL ;	//Temporary REAL
  dTmp : DINT ;	//Temporary DINT (free for general use)
  RetValInt : INT ;	//return value
END_VAR
BEGIN
NETWORK
TITLE =General

      SET   ;
// Simulation ---------------------------------------------------------------
      A     DB4281.DBX 1357.7;
      CC    FB  4289; // "U128Sim"
      A     DB4281.DBX   17.3;
      =     DB4281.DBX 1357.7; //Help bit for simulation

// get unit number ----------------------------------------------------------
      L     DB4280.DBW    0;
      T     #UnitNo;

// CIP ----------------------------------------------------------------------
      L     DB4281.DBD   54;
      L     0;
      <D    ;
      =     #CIP;

// emergency OK -------------------------------------------------------------
      A     DB4285.DBX   27.0; //Emergency Stop OK
      =     #EStopOK;

// Write Unit in Maintenance ------------------------------------------------

      AN    DB4281.DBX   69.7;
      =     #UNIM;

// emergency and maintenance OK ---------------------------------------------
      A     #EStopOK;
      A     #UNIM;
      =     #GenRel;

// communication ------------------------------------------------------------
      UC    FB  4285; // U128Com

NETWORK
TITLE =Analog Inputs

      NOP   0;

// ----------------------------------------------------------
// C_AnI01 spare
// ----------------------------------------------------------
      L     DB4281.DBD 1118; // !!! insert correct SFM !!!
      T     DB5283.DBD  238;

      SET   ;
      =     DB5283.DBX  141.5;

// ----------------------------------------------------------
// C_AnI002 spare
// ----------------------------------------------------------
      L     DB4281.DBD 1118; // !!! insert correct SFM !!!
      T     DB5283.DBD  358;

      SET   ;
      =     DB5283.DBX  261.5;

// ----------------------------------------------------------
// AnI03 spare
// ----------------------------------------------------------
      L     DB4281.DBD 1118; // !!! insert correct SFM !!!
      T     DB5283.DBD  478;

      SET   ;
      =     DB5283.DBX  381.5;

NETWORK
TITLE =Universal Value

      NOP   0;

// ----------------------------------------------------------
// unv001 Process Status
// ----------------------------------------------------------
// process value to UnV
//      L     0.000000e+000
//      T     "U128UnVD".unv001.ValExt

// ----------------------------------------------------------
// unv002 Universal Value 02
// ----------------------------------------------------------
// process value to UnV
//      L     0.000000e+000
//      T     "U128UnVD".unv002.ValExt

// ----------------------------------------------------------
// unv003 Druck Sollwert
// ----------------------------------------------------------
// process value to UnV
//      L     0.000000e+000
//      T     "U128UnVD".unv003.ValExt

// ----------------------------------------------------------
// unv004 Universal Value 04
// ----------------------------------------------------------
// process value to UnV
//      L     0.000000e+000
//      T     "U128UnVD".unv004.ValExt

NETWORK
TITLE =Special Input

      NOP   0;

// ----------------------------------------------------------
// SpI01 spare
// ----------------------------------------------------------
      SET   ;
      =     DB5281.DBX   81.4;
      =     DB5281.DBX   81.5;

// ----------------------------------------------------------
// SpI02 spare
// ----------------------------------------------------------
      SET   ;
      =     DB5281.DBX  141.4;
      =     DB5281.DBX  141.5;

// ----------------------------------------------------------
// SpI03 spare
// ----------------------------------------------------------
      SET   ;
      =     DB5281.DBX  201.4;
      =     DB5281.DBX  201.5;

// ----------------------------------------------------------
// SpI04 spare
// ----------------------------------------------------------
      SET   ;
      =     DB5281.DBX  261.4;
      =     DB5281.DBX  261.5;

NETWORK
TITLE =Messages

      NOP   0;

// ----------------------------------------------------------
// msg001 Message 01
// ----------------------------------------------------------
      SET   ;
      R     DB5287.DBX   80.7;
      =     DB5287.DBX   81.4;

      CLR   ;
      =     DB5287.DBX   82.7;

// ----------------------------------------------------------
// msg002 Message 02
// ----------------------------------------------------------
      SET   ;
      R     DB5287.DBX  140.7;
      =     DB5287.DBX  141.4;

      CLR   ;
      =     DB5287.DBX  142.7;

// ----------------------------------------------------------
// msg003 Message 03
// ----------------------------------------------------------
      SET   ;
      R     DB5287.DBX  200.7;
      =     DB5287.DBX  201.4;

      CLR   ;
      =     DB5287.DBX  202.7;

NETWORK
TITLE =PID controller

      NOP   0;

// ----------------------------------------------------------
// PID01 spare
// ----------------------------------------------------------
// starting value -----------------------
//A     "U128ActD".Act.OutI // !!! insert correct Act !!!
      A     #GenRel;
      CLR   ;
      =     DB5286.DBX  203.2;
      =     DB5286.DBX  203.5;

// enable alarm -------------------------
      A     DB5286.DBX  203.5;
      A     DB5286.DBX  201.4;
      AN    DB5286.DBX  203.1;
      AN    DB5286.DBX  203.3;
      AN    DB5286.DBX  203.4;
      =     DB5286.DBX  203.0;

// setpoint to controller ---------------
      L     DB4281.DBD 1118; // !!! insert correct SFM !!!
      T     DB5286.DBD  234;

// static value to controller ----------
      L     DB4281.DBD 1118; // !!! insert correct SFM !!!
      T     DB5286.DBD  238;

// process value to controller ----------
      L     DB5283.DBD   26; // !!! insert correct AnI !!!
      T     DB5286.DBD  254;

// low/high value to controller ---------
      L     DB5283.DBD   30; // !!! insert correct AnI !!!
      T     DB5286.DBD  218;

      L     DB5283.DBD   34; // !!! insert correct AnI !!!
      T     DB5286.DBD  222;

NETWORK
TITLE =Sequence organisation

      CLR   ;
      =     M    122.2;

// SFM supply ----------------------------------------------------------------

// analog value to SFM spare -----------------------
      L     DB5283.DBD  146;
      T     DB4281.DBD 1122; // !!! insert correct SFM !!!

// analog value to SFM spare -----------------------
      L     DB5283.DBD  266;
      T     DB4281.DBD 1122; // !!! insert correct SFM !!!

// analog value to SFM spare -----------------------
      L     DB5283.DBD  386;
      T     DB4281.DBD 1122; // !!! insert correct SFM !!!

// sequencer ----------------------------------------------------------------
      A     DB4283.DBX   43.1;
      S     DB4283.DBX   97.3;

      CALL FC    40 (
           UnitNo                   := #UnitNo);

NETWORK
TITLE =Auto / Manual

      SET   ;
      AN    M    122.2;
      JC    MODE;
      AN    M    120.1;


// assign PID mode
      S     DB5286.DBX  201.4;
      S     DB5286.DBX  201.5;


MODE: SET   ;

END_FUNCTION_BLOCK

FUNCTION_BLOCK FB 4290
TITLE =U129: Planung Transfer B6F
FAMILY : BOTEC_F1
NAME : U129A
VERSION : 2.1


VAR_TEMP
  EStopOK : BOOL ;	//auxiliary flag
  CIP : BOOL ;	//CIP Program Selected
  xTmp : BOOL ;	//Temporary Bool(free for general use)
  DummyBool : BOOL ;	//Temporary Bool(free for general use)
  UnitNo : INT ;	//unit number
  UnitFB : INT ;	//unit expansion FB number
  rTmp : REAL ;	//Temporary REAL (free for general use)
  iTmp : INT ;	//Temporary INT (free for general use)
  DummyInt : INT ;	//Temporary INT (free for general use)
  dTmp : DINT ;	//Temporary DINT (free for general use)
END_VAR
BEGIN
NETWORK
TITLE =general

      CLR   ;
      =     #xTmp;
      =     #EStopOK;

      L     DB4290.DBW    0;
      T     #UnitNo;
      L     DB4290.DBW    2;
      T     #UnitFB;

NETWORK
TITLE =analog inputs

      NOP   0;
// C_AnI01 AnI 001 spare
      CALL FC    24 (
           UnitNo                   := #UnitNo,
           AnIRec                   := DB5293.C_AnI01,
           ValPer                   := #DummyInt);

// C_AnI002 AnI 002 spare
      CALL FC    24 (
           UnitNo                   := #UnitNo,
           AnIRec                   := DB5293.C_AnI002,
           ValPer                   := #DummyInt);

// AnI03 AnI 003 spare
      CALL FC    24 (
           UnitNo                   := #UnitNo,
           AnIRec                   := DB5293.AnI03,
           ValPer                   := #DummyInt);

NETWORK
TITLE =Universal value

      NOP   0;
// unv001 UnV 001 Process Status
      CALL FC    27 (
           UnitNo                   := #UnitNo,
           UnVRec                   := DB5295.unv001,
           ValExt                   := DB5295.DBD  234);

// unv002 UnV 002 Universal Value 02
      CALL FC    27 (
           UnitNo                   := #UnitNo,
           UnVRec                   := DB5295.unv002,
           ValExt                   := DB5295.DBD  362);

// unv003 UnV 003 Druck Sollwert
      CALL FC    27 (
           UnitNo                   := #UnitNo,
           UnVRec                   := DB5295.unv003,
           ValExt                   := DB5295.DBD  490);

// unv004 UnV 004 Universal Value 04
      CALL FC    27 (
           UnitNo                   := #UnitNo,
           UnVRec                   := DB5295.unv004,
           ValExt                   := DB5295.DBD  618);

NETWORK
TITLE =special inputs

      NOP   0;
// SpI01 SpI 001 spare
      CALL FC    14 (
           UnitNo                   := #UnitNo,
           SpIRec                   := DB5291.SpI01,
           SpIBit                   := #DummyBool);

// SpI02 SpI 002 spare
      CALL FC    14 (
           UnitNo                   := #UnitNo,
           SpIRec                   := DB5291.SpI02,
           SpIBit                   := #DummyBool);

// SpI03 SpI 003 spare
      CALL FC    14 (
           UnitNo                   := #UnitNo,
           SpIRec                   := DB5291.SpI03,
           SpIBit                   := #DummyBool);

// SpI04 SpI 004 spare
      CALL FC    14 (
           UnitNo                   := #UnitNo,
           SpIRec                   := DB5291.SpI04,
           SpIBit                   := #DummyBool);

NETWORK
TITLE =messages

      NOP   0;
// msg001 Msg 001 Message 01
      CALL FC    16 (
           UnitNo                   := #UnitNo,
           MsgRec                   := DB5297.msg001,
           MsgBit                   := DB5297.DBX   82.7);

// msg002 Msg 002 Message 02
      CALL FC    16 (
           UnitNo                   := #UnitNo,
           MsgRec                   := DB5297.msg002,
           MsgBit                   := DB5297.DBX  142.7);

// msg003 Msg 003 Message 03
      CALL FC    16 (
           UnitNo                   := #UnitNo,
           MsgRec                   := DB5297.msg003,
           MsgBit                   := DB5297.DBX  202.7);

NETWORK
TITLE =controllers

      NOP   0;
// PID01 PID 001 spare
      CALL FC    55 (
           UnitNo                   := #UnitNo,
           PIDRec                   := DB5296.PID01,
           SpExt                    := DB5296.DBD  234,
           PVal                     := DB5296.DBD  254,
           OPer                     := #DummyInt);

NETWORK
TITLE =unit supply

      UC    FB [#UnitFB];
END_FUNCTION_BLOCK

FUNCTION_BLOCK FB 4291
TITLE =U129: Planung Transfer B6F
FAMILY : BOTEC_F1
NAME : U129E
VERSION : 1.2


VAR_TEMP
  CIP : BOOL ;	//CIP active
  UNIM : BOOL ;	//Unit Not In Maintenance
  GenRel : BOOL ;	//general OK (emergency and maintenance OK)
  EStopOK : BOOL ;	//emergency OK
  UnitNo : INT ;	//unit number
  xTmp : BOOL ;	//Temporary Bool
  iTmp : INT ;	//Temporary INT
  rTmp : REAL ;	//Temporary REAL
  dTmp : DINT ;	//Temporary DINT (free for general use)
  RetValInt : INT ;	//return value
END_VAR
BEGIN
NETWORK
TITLE =General

      SET   ;
// Simulation ---------------------------------------------------------------
      A     DB4291.DBX 1357.7;
      CC    FB  4299; // "U129Sim"
      A     DB4291.DBX   17.3;
      =     DB4291.DBX 1357.7; //Help bit for simulation

// get unit number ----------------------------------------------------------
      L     DB4290.DBW    0;
      T     #UnitNo;

// CIP ----------------------------------------------------------------------
      L     DB4291.DBD   54;
      L     0;
      <D    ;
      =     #CIP;

// emergency OK -------------------------------------------------------------
      A     DB4295.DBX   27.0; //Emergency Stop OK
      =     #EStopOK;

// Write Unit in Maintenance ------------------------------------------------

      AN    DB4291.DBX   69.7;
      =     #UNIM;

// emergency and maintenance OK ---------------------------------------------
      A     #EStopOK;
      A     #UNIM;
      =     #GenRel;

// communication ------------------------------------------------------------
      UC    FB  4295; // U129Com

NETWORK
TITLE =Analog Inputs

      NOP   0;

// ----------------------------------------------------------
// C_AnI01 spare
// ----------------------------------------------------------
      L     DB4291.DBD 1118; // !!! insert correct SFM !!!
      T     DB5293.DBD  238;

      SET   ;
      =     DB5293.DBX  141.5;

// ----------------------------------------------------------
// C_AnI002 spare
// ----------------------------------------------------------
      L     DB4291.DBD 1118; // !!! insert correct SFM !!!
      T     DB5293.DBD  358;

      SET   ;
      =     DB5293.DBX  261.5;

// ----------------------------------------------------------
// AnI03 spare
// ----------------------------------------------------------
      L     DB4291.DBD 1118; // !!! insert correct SFM !!!
      T     DB5293.DBD  478;

      SET   ;
      =     DB5293.DBX  381.5;

NETWORK
TITLE =Universal Value

      NOP   0;

// ----------------------------------------------------------
// unv001 Process Status
// ----------------------------------------------------------
// process value to UnV
//      L     0.000000e+000
//      T     "U129UnVD".unv001.ValExt

// ----------------------------------------------------------
// unv002 Universal Value 02
// ----------------------------------------------------------
// process value to UnV
//      L     0.000000e+000
//      T     "U129UnVD".unv002.ValExt

// ----------------------------------------------------------
// unv003 Druck Sollwert
// ----------------------------------------------------------
// process value to UnV
//      L     0.000000e+000
//      T     "U129UnVD".unv003.ValExt

// ----------------------------------------------------------
// unv004 Universal Value 04
// ----------------------------------------------------------
// process value to UnV
//      L     0.000000e+000
//      T     "U129UnVD".unv004.ValExt

NETWORK
TITLE =Special Input

      NOP   0;

// ----------------------------------------------------------
// SpI01 spare
// ----------------------------------------------------------
      SET   ;
      =     DB5291.DBX   81.4;
      =     DB5291.DBX   81.5;

// ----------------------------------------------------------
// SpI02 spare
// ----------------------------------------------------------
      SET   ;
      =     DB5291.DBX  141.4;
      =     DB5291.DBX  141.5;

// ----------------------------------------------------------
// SpI03 spare
// ----------------------------------------------------------
      SET   ;
      =     DB5291.DBX  201.4;
      =     DB5291.DBX  201.5;

// ----------------------------------------------------------
// SpI04 spare
// ----------------------------------------------------------
      SET   ;
      =     DB5291.DBX  261.4;
      =     DB5291.DBX  261.5;

NETWORK
TITLE =Messages

      NOP   0;

// ----------------------------------------------------------
// msg001 Message 01
// ----------------------------------------------------------
      SET   ;
      R     DB5297.DBX   80.7;
      =     DB5297.DBX   81.4;

      CLR   ;
      =     DB5297.DBX   82.7;

// ----------------------------------------------------------
// msg002 Message 02
// ----------------------------------------------------------
      SET   ;
      R     DB5297.DBX  140.7;
      =     DB5297.DBX  141.4;

      CLR   ;
      =     DB5297.DBX  142.7;

// ----------------------------------------------------------
// msg003 Message 03
// ----------------------------------------------------------
      SET   ;
      R     DB5297.DBX  200.7;
      =     DB5297.DBX  201.4;

      CLR   ;
      =     DB5297.DBX  202.7;

NETWORK
TITLE =PID controller

      NOP   0;

// ----------------------------------------------------------
// PID01 spare
// ----------------------------------------------------------
// starting value -----------------------
//A     "U129ActD".Act.OutI // !!! insert correct Act !!!
      A     #GenRel;
      CLR   ;
      =     DB5296.DBX  203.2;
      =     DB5296.DBX  203.5;

// enable alarm -------------------------
      A     DB5296.DBX  203.5;
      A     DB5296.DBX  201.4;
      AN    DB5296.DBX  203.1;
      AN    DB5296.DBX  203.3;
      AN    DB5296.DBX  203.4;
      =     DB5296.DBX  203.0;

// setpoint to controller ---------------
      L     DB4291.DBD 1118; // !!! insert correct SFM !!!
      T     DB5296.DBD  234;

// static value to controller ----------
      L     DB4291.DBD 1118; // !!! insert correct SFM !!!
      T     DB5296.DBD  238;

// process value to controller ----------
      L     DB5293.DBD   26; // !!! insert correct AnI !!!
      T     DB5296.DBD  254;

// low/high value to controller ---------
      L     DB5293.DBD   30; // !!! insert correct AnI !!!
      T     DB5296.DBD  218;

      L     DB5293.DBD   34; // !!! insert correct AnI !!!
      T     DB5296.DBD  222;

NETWORK
TITLE =Sequence organisation

      CLR   ;
      =     M    122.2;

// SFM supply ----------------------------------------------------------------

// analog value to SFM spare -----------------------
      L     DB5293.DBD  146;
      T     DB4291.DBD 1122; // !!! insert correct SFM !!!

// analog value to SFM spare -----------------------
      L     DB5293.DBD  266;
      T     DB4291.DBD 1122; // !!! insert correct SFM !!!

// analog value to SFM spare -----------------------
      L     DB5293.DBD  386;
      T     DB4291.DBD 1122; // !!! insert correct SFM !!!

// sequencer ----------------------------------------------------------------
      A     DB4293.DBX   43.1;
      S     DB4293.DBX   97.3;

      CALL FC    40 (
           UnitNo                   := #UnitNo);

NETWORK
TITLE =Auto / Manual

      SET   ;
      AN    M    122.2;
      JC    MODE;
      AN    M    120.1;


// assign PID mode
      S     DB5296.DBX  201.4;
      S     DB5296.DBX  201.5;


MODE: SET   ;

END_FUNCTION_BLOCK

FUNCTION_BLOCK FB 4300
TITLE =U130: Planung Transfer H6F
FAMILY : BOTEC_F1
NAME : U130A
VERSION : 2.1


VAR_TEMP
  EStopOK : BOOL ;	//auxiliary flag
  CIP : BOOL ;	//CIP Program Selected
  xTmp : BOOL ;	//Temporary Bool(free for general use)
  DummyBool : BOOL ;	//Temporary Bool(free for general use)
  UnitNo : INT ;	//unit number
  UnitFB : INT ;	//unit expansion FB number
  rTmp : REAL ;	//Temporary REAL (free for general use)
  iTmp : INT ;	//Temporary INT (free for general use)
  DummyInt : INT ;	//Temporary INT (free for general use)
  dTmp : DINT ;	//Temporary DINT (free for general use)
END_VAR
BEGIN
NETWORK
TITLE =general

      CLR   ;
      =     #xTmp;
      =     #EStopOK;

      L     DB4300.DBW    0;
      T     #UnitNo;
      L     DB4300.DBW    2;
      T     #UnitFB;

NETWORK
TITLE =analog inputs

      NOP   0;
// C_AnI01 AnI 001 spare
      CALL FC    24 (
           UnitNo                   := #UnitNo,
           AnIRec                   := DB5303.C_AnI01,
           ValPer                   := #DummyInt);

// C_AnI002 AnI 002 spare
      CALL FC    24 (
           UnitNo                   := #UnitNo,
           AnIRec                   := DB5303.C_AnI002,
           ValPer                   := #DummyInt);

// AnI03 AnI 003 spare
      CALL FC    24 (
           UnitNo                   := #UnitNo,
           AnIRec                   := DB5303.AnI03,
           ValPer                   := #DummyInt);

NETWORK
TITLE =Universal value

      NOP   0;
// unv001 UnV 001 Process Status
      CALL FC    27 (
           UnitNo                   := #UnitNo,
           UnVRec                   := DB5305.unv001,
           ValExt                   := DB5305.DBD  234);

// unv002 UnV 002 Universal Value 02
      CALL FC    27 (
           UnitNo                   := #UnitNo,
           UnVRec                   := DB5305.unv002,
           ValExt                   := DB5305.DBD  362);

// unv003 UnV 003 Druck Sollwert
      CALL FC    27 (
           UnitNo                   := #UnitNo,
           UnVRec                   := DB5305.unv003,
           ValExt                   := DB5305.DBD  490);

// unv004 UnV 004 Universal Value 04
      CALL FC    27 (
           UnitNo                   := #UnitNo,
           UnVRec                   := DB5305.unv004,
           ValExt                   := DB5305.DBD  618);

NETWORK
TITLE =special inputs

      NOP   0;
// SpI01 SpI 001 spare
      CALL FC    14 (
           UnitNo                   := #UnitNo,
           SpIRec                   := DB5301.SpI01,
           SpIBit                   := #DummyBool);

// SpI02 SpI 002 spare
      CALL FC    14 (
           UnitNo                   := #UnitNo,
           SpIRec                   := DB5301.SpI02,
           SpIBit                   := #DummyBool);

// SpI03 SpI 003 spare
      CALL FC    14 (
           UnitNo                   := #UnitNo,
           SpIRec                   := DB5301.SpI03,
           SpIBit                   := #DummyBool);

// SpI04 SpI 004 spare
      CALL FC    14 (
           UnitNo                   := #UnitNo,
           SpIRec                   := DB5301.SpI04,
           SpIBit                   := #DummyBool);

NETWORK
TITLE =messages

      NOP   0;
// msg001 Msg 001 Message 01
      CALL FC    16 (
           UnitNo                   := #UnitNo,
           MsgRec                   := DB5307.msg001,
           MsgBit                   := DB5307.DBX   82.7);

// msg002 Msg 002 Message 02
      CALL FC    16 (
           UnitNo                   := #UnitNo,
           MsgRec                   := DB5307.msg002,
           MsgBit                   := DB5307.DBX  142.7);

// msg003 Msg 003 Message 03
      CALL FC    16 (
           UnitNo                   := #UnitNo,
           MsgRec                   := DB5307.msg003,
           MsgBit                   := DB5307.DBX  202.7);

NETWORK
TITLE =controllers

      NOP   0;
// PID01 PID 001 spare
      CALL FC    55 (
           UnitNo                   := #UnitNo,
           PIDRec                   := DB5306.PID01,
           SpExt                    := DB5306.DBD  234,
           PVal                     := DB5306.DBD  254,
           OPer                     := #DummyInt);

NETWORK
TITLE =unit supply

      UC    FB [#UnitFB];
END_FUNCTION_BLOCK

FUNCTION_BLOCK FB 4301
TITLE =U130: Planung Transfer H6F
FAMILY : BOTEC_F1
NAME : U130E
VERSION : 1.2


VAR_TEMP
  CIP : BOOL ;	//CIP active
  UNIM : BOOL ;	//Unit Not In Maintenance
  GenRel : BOOL ;	//general OK (emergency and maintenance OK)
  EStopOK : BOOL ;	//emergency OK
  UnitNo : INT ;	//unit number
  xTmp : BOOL ;	//Temporary Bool
  iTmp : INT ;	//Temporary INT
  rTmp : REAL ;	//Temporary REAL
  dTmp : DINT ;	//Temporary DINT (free for general use)
  RetValInt : INT ;	//return value
END_VAR
BEGIN
NETWORK
TITLE =General

      SET   ;
// Simulation ---------------------------------------------------------------
      A     DB4301.DBX 1357.7;
      CC    FB  4309; // "U130Sim"
      A     DB4301.DBX   17.3;
      =     DB4301.DBX 1357.7; //Help bit for simulation

// get unit number ----------------------------------------------------------
      L     DB4300.DBW    0;
      T     #UnitNo;

// CIP ----------------------------------------------------------------------
      L     DB4301.DBD   54;
      L     0;
      <D    ;
      =     #CIP;

// emergency OK -------------------------------------------------------------
      A     DB4305.DBX   27.0; //Emergency Stop OK
      =     #EStopOK;

// Write Unit in Maintenance ------------------------------------------------

      AN    DB4301.DBX   69.7;
      =     #UNIM;

// emergency and maintenance OK ---------------------------------------------
      A     #EStopOK;
      A     #UNIM;
      =     #GenRel;

// communication ------------------------------------------------------------
      UC    FB  4305; // U130Com

NETWORK
TITLE =Analog Inputs

      NOP   0;

// ----------------------------------------------------------
// C_AnI01 spare
// ----------------------------------------------------------
      L     DB4301.DBD 1118; // !!! insert correct SFM !!!
      T     DB5303.DBD  238;

      SET   ;
      =     DB5303.DBX  141.5;

// ----------------------------------------------------------
// C_AnI002 spare
// ----------------------------------------------------------
      L     DB4301.DBD 1118; // !!! insert correct SFM !!!
      T     DB5303.DBD  358;

      SET   ;
      =     DB5303.DBX  261.5;

// ----------------------------------------------------------
// AnI03 spare
// ----------------------------------------------------------
      L     DB4301.DBD 1118; // !!! insert correct SFM !!!
      T     DB5303.DBD  478;

      SET   ;
      =     DB5303.DBX  381.5;

NETWORK
TITLE =Universal Value

      NOP   0;

// ----------------------------------------------------------
// unv001 Process Status
// ----------------------------------------------------------
// process value to UnV
//      L     0.000000e+000
//      T     "U130UnVD".unv001.ValExt

// ----------------------------------------------------------
// unv002 Universal Value 02
// ----------------------------------------------------------
// process value to UnV
//      L     0.000000e+000
//      T     "U130UnVD".unv002.ValExt

// ----------------------------------------------------------
// unv003 Druck Sollwert
// ----------------------------------------------------------
// process value to UnV
//      L     0.000000e+000
//      T     "U130UnVD".unv003.ValExt

// ----------------------------------------------------------
// unv004 Universal Value 04
// ----------------------------------------------------------
// process value to UnV
//      L     0.000000e+000
//      T     "U130UnVD".unv004.ValExt

NETWORK
TITLE =Special Input

      NOP   0;

// ----------------------------------------------------------
// SpI01 spare
// ----------------------------------------------------------
      SET   ;
      =     DB5301.DBX   81.4;
      =     DB5301.DBX   81.5;

// ----------------------------------------------------------
// SpI02 spare
// ----------------------------------------------------------
      SET   ;
      =     DB5301.DBX  141.4;
      =     DB5301.DBX  141.5;

// ----------------------------------------------------------
// SpI03 spare
// ----------------------------------------------------------
      SET   ;
      =     DB5301.DBX  201.4;
      =     DB5301.DBX  201.5;

// ----------------------------------------------------------
// SpI04 spare
// ----------------------------------------------------------
      SET   ;
      =     DB5301.DBX  261.4;
      =     DB5301.DBX  261.5;

NETWORK
TITLE =Messages

      NOP   0;

// ----------------------------------------------------------
// msg001 Message 01
// ----------------------------------------------------------
      SET   ;
      R     DB5307.DBX   80.7;
      =     DB5307.DBX   81.4;

      CLR   ;
      =     DB5307.DBX   82.7;

// ----------------------------------------------------------
// msg002 Message 02
// ----------------------------------------------------------
      SET   ;
      R     DB5307.DBX  140.7;
      =     DB5307.DBX  141.4;

      CLR   ;
      =     DB5307.DBX  142.7;

// ----------------------------------------------------------
// msg003 Message 03
// ----------------------------------------------------------
      SET   ;
      R     DB5307.DBX  200.7;
      =     DB5307.DBX  201.4;

      CLR   ;
      =     DB5307.DBX  202.7;

NETWORK
TITLE =PID controller

      NOP   0;

